Yaskawa INFORM job: DEMO_ROOF_UPPER_0625_3.JBI

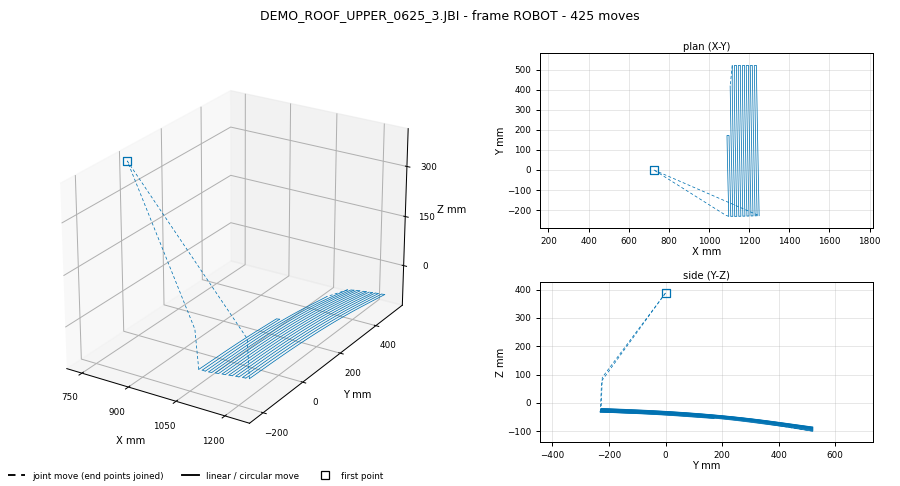
[picture p0: tool path of DEMO_ROOF_UPPER_0625_3.JBI in frame ROBOT, 425 of 425 moves have a stored position in this frame; points joined in program order, loops and branches not executed]
/JOB
//NAME DEMO_ROOF_UPPER_0625_3
//POS
///NPOS 425,0,0,0,0,0
///TOOL 0
///USER 0
///POSTYPE ROBOT
///RECTAN
///RCONF 1,0,0,0,0,0,0,0,0,0,0,0,0,0,0,0,0,0,0,0,0,0,0,0
C00000=725.000,0.000,388.500,-180.000,-0.000,0.000
///USER 0
///POSTYPE ROBOT
///RECTAN
C00001=1240.342,-223.716,89.889,177.727,-4.742,1.457
C00002=1249.517,-227.840,-19.446,177.737,-4.746,1.344
C00003=1247.381,-125.286,-23.774,177.737,-4.746,1.344
C00004=1246.860,-99.191,-24.873,177.524,-4.614,1.344
C00005=1246.366,-74.184,-26.020,177.315,-4.486,1.346
C00006=1245.874,-49.099,-27.262,177.100,-4.359,1.346
C00007=1245.386,-24.019,-28.598,176.878,-4.234,1.350
C00008=1244.921,0.054,-29.974,176.660,-4.119,1.352
C00009=1244.459,24.123,-31.441,176.435,-4.011,1.354
C00010=1244.000,48.187,-33.000,176.203,-3.911,1.356
C00011=1243.563,71.245,-34.588,175.975,-3.823,1.358
C00012=1243.128,94.298,-36.268,175.738,-3.746,1.364
C00013=1242.714,116.348,-37.962,175.506,-3.682,1.369
C00014=1242.302,138.394,-39.747,175.266,-3.631,1.372
C00015=1241.895,160.355,-41.616,175.018,-3.590,1.379
C00016=1241.506,181.391,-43.496,174.774,-3.563,1.388
C00017=1241.119,202.423,-45.465,174.522,-3.547,1.395
C00018=1240.735,223.453,-47.526,174.262,-3.543,1.405
C00019=1240.353,244.477,-49.679,173.998,-3.551,1.415
C00020=1239.993,264.406,-51.810,173.743,-3.570,1.430
C00021=1239.632,284.422,-54.040,173.482,-3.603,1.446
C00022=1239.273,304.436,-56.359,173.220,-3.652,1.464
C00023=1238.915,324.446,-58.768,172.960,-3.719,1.487
C00024=1238.558,344.452,-61.261,172.707,-3.804,1.516
C00025=1238.185,365.319,-63.950,172.464,-3.916,1.544
C00026=1237.775,388.282,-67.000,172.236,-4.061,1.575
C00027=1237.234,418.731,-71.176,172.012,-4.269,1.516
C00028=1235.598,520.410,-85.296,172.012,-4.269,1.516
C00029=1225.496,520.130,-86.161,172.024,-4.292,1.352
C00030=1227.173,414.926,-71.461,172.041,-4.257,1.444
C00031=1227.647,388.013,-67.749,172.243,-4.076,1.464
C00032=1228.055,365.054,-64.671,172.469,-3.926,1.465
C00033=1228.426,344.191,-61.961,172.711,-3.812,1.457
C00034=1228.783,324.187,-59.451,172.962,-3.723,1.446
C00035=1229.140,304.179,-57.031,173.222,-3.656,1.435
C00036=1229.498,284.168,-54.703,173.484,-3.606,1.425
C00037=1229.858,264.154,-52.466,173.744,-3.572,1.416
C00038=1230.218,244.226,-50.331,173.999,-3.552,1.409
C00039=1230.600,223.202,-48.173,174.262,-3.543,1.402
C00040=1230.984,202.174,-46.113,174.522,-3.547,1.397
C00041=1231.370,181.143,-44.146,174.773,-3.563,1.393
C00042=1231.759,160.106,-42.271,175.017,-3.589,1.390
C00043=1232.168,138.146,-40.407,175.265,-3.629,1.388
C00044=1232.580,116.100,-38.632,175.504,-3.681,1.387
C00045=1232.995,94.051,-36.947,175.737,-3.744,1.387
C00046=1233.430,70.997,-35.281,175.973,-3.821,1.388
C00047=1233.868,47.939,-33.708,176.201,-3.908,1.389
C00048=1234.328,23.876,-32.165,176.433,-4.009,1.390
C00049=1234.792,-0.193,-30.716,176.657,-4.117,1.392
C00050=1235.258,-24.267,-29.361,176.875,-4.232,1.394
C00051=1235.748,-49.347,-28.046,177.096,-4.356,1.396
C00052=1236.242,-74.432,-26.825,177.311,-4.484,1.398
C00053=1236.738,-99.438,-25.702,177.519,-4.611,1.401
C00054=1237.260,-125.533,-24.625,177.731,-4.744,1.408
C00055=1239.404,-228.090,-20.387,177.730,-4.743,1.421
C00056=1229.270,-228.359,-21.330,177.730,-4.743,1.425
C00057=1227.118,-125.798,-25.478,177.786,-4.870,1.350
C00058=1226.593,-99.702,-26.531,177.573,-4.744,1.353
C00059=1226.094,-74.695,-27.633,177.364,-4.620,1.354
C00060=1225.598,-49.609,-28.830,177.149,-4.498,1.356
C00061=1225.106,-24.527,-30.124,176.927,-4.377,1.357
C00062=1224.638,-0.451,-31.460,176.705,-4.267,1.363
C00063=1224.171,23.619,-32.889,176.477,-4.162,1.363
C00064=1223.729,46.685,-34.351,176.252,-4.070,1.369
C00065=1223.289,69.746,-35.904,176.019,-3.988,1.374
C00066=1222.851,92.801,-37.553,175.778,-3.915,1.379
C00067=1222.434,114.852,-39.224,175.541,-3.856,1.382
C00068=1222.021,136.900,-40.986,175.295,-3.808,1.391
C00069=1221.611,158.862,-42.838,175.043,-3.773,1.400
C00070=1221.220,179.899,-44.706,174.793,-3.751,1.405
C00071=1220.833,200.933,-46.665,174.536,-3.740,1.418
C00072=1220.447,221.963,-48.722,174.270,-3.742,1.425
C00073=1220.083,241.991,-50.773,174.013,-3.754,1.441
C00074=1219.721,261.920,-52.903,173.752,-3.778,1.453
C00075=1219.361,281.936,-55.137,173.484,-3.816,1.473
C00076=1219.002,301.949,-57.466,173.213,-3.868,1.492
C00077=1218.644,321.959,-59.890,172.942,-3.938,1.516
C00078=1218.290,341.844,-62.393,172.680,-4.027,1.546
C00079=1217.934,361.836,-64.998,172.432,-4.137,1.577
C00080=1217.544,383.804,-67.956,172.199,-4.283,1.605
C00081=1217.087,409.726,-71.548,172.001,-4.478,1.535
C00082=1215.344,520.125,-87.069,171.946,-4.534,1.543
C00083=1205.181,520.128,-88.023,171.968,-4.573,1.268
C00084=1206.771,418.484,-73.649,171.887,-4.817,1.451
C00085=1207.039,402.544,-71.393,171.980,-4.698,1.499
C00086=1207.480,377.609,-67.929,172.188,-4.502,1.531
C00087=1207.852,356.628,-65.100,172.432,-4.355,1.529
C00088=1208.208,336.632,-62.495,172.695,-4.241,1.517
C00089=1208.562,316.743,-59.999,172.970,-4.151,1.502
C00090=1208.902,297.725,-57.703,173.236,-4.082,1.487
C00091=1209.244,278.705,-55.496,173.500,-4.029,1.474
C00092=1209.605,258.687,-53.270,173.774,-3.986,1.462
C00093=1209.968,238.756,-51.147,174.040,-3.957,1.452
C00094=1210.333,218.726,-49.107,174.303,-3.939,1.443
C00095=1210.703,198.691,-47.158,174.560,-3.933,1.436
C00096=1211.092,177.657,-45.208,174.822,-3.938,1.429
C00097=1211.484,156.617,-43.353,175.077,-3.956,1.424
C00098=1211.876,135.651,-41.597,175.322,-3.985,1.420
C00099=1212.291,113.603,-39.846,175.572,-4.027,1.417
C00100=1212.710,91.550,-38.190,175.815,-4.081,1.415
C00101=1213.129,69.491,-36.627,176.049,-4.146,1.414
C00102=1213.572,46.429,-35.087,176.287,-4.225,1.413
C00103=1214.017,23.362,-33.642,176.515,-4.312,1.413
C00104=1214.485,-0.710,-32.229,176.746,-4.411,1.413
C00105=1214.956,-24.788,-30.913,176.969,-4.517,1.413
C00106=1215.450,-49.871,-29.640,177.193,-4.632,1.413
C00107=1215.949,-74.960,-28.463,177.409,-4.751,1.413
C00108=1216.450,-99.968,-27.384,177.617,-4.870,1.414
C00109=1216.979,-126.065,-26.352,177.828,-4.992,1.419
C00110=1219.138,-228.629,-22.291,177.826,-4.991,1.444
C00111=1209.008,-228.900,-23.270,177.826,-4.991,1.443
C00112=1206.841,-126.333,-27.248,177.879,-5.116,1.364
C00113=1206.310,-100.234,-28.259,177.669,-5.000,1.368
C00114=1205.806,-75.226,-29.318,177.461,-4.886,1.369
C00115=1205.305,-50.136,-30.474,177.243,-4.772,1.374
C00116=1204.828,-26.050,-31.675,177.025,-4.666,1.379
C00117=1204.354,-1.971,-32.970,176.800,-4.564,1.383
C00118=1203.883,22.103,-34.360,176.566,-4.469,1.387
C00119=1203.437,45.172,-35.787,176.333,-4.386,1.393
C00120=1202.992,68.236,-37.309,176.092,-4.312,1.401
C00121=1202.570,90.296,-38.858,175.853,-4.252,1.406
C00122=1202.151,112.351,-40.500,175.605,-4.202,1.416
C00123=1201.754,133.325,-42.153,175.362,-4.166,1.425
C00124=1201.358,154.370,-43.902,175.109,-4.140,1.431
C00125=1200.965,175.412,-45.745,174.849,-4.127,1.446
C00126=1200.593,195.451,-47.592,174.595,-4.125,1.458
C00127=1200.223,215.487,-49.529,174.332,-4.134,1.469
C00128=1199.857,235.428,-51.549,174.065,-4.155,1.487
C00129=1199.492,255.451,-53.673,173.791,-4.189,1.502
C00130=1199.148,274.476,-55.782,173.525,-4.233,1.522
C00131=1198.805,293.499,-57.981,173.254,-4.290,1.542
C00132=1198.467,312.407,-60.256,172.981,-4.359,1.566
C00133=1198.129,331.416,-62.637,172.707,-4.443,1.595
C00134=1197.791,350.423,-65.107,172.439,-4.546,1.631
C00135=1197.436,370.419,-67.800,172.178,-4.681,1.666
C00136=1197.033,393.235,-70.973,171.954,-4.868,1.663
C00137=1196.606,418.506,-74.570,171.896,-5.210,0.598
C00138=1196.859,520.156,-88.981,171.896,-5.210,0.598
C00139=1185.350,520.147,-90.183,171.840,-5.121,1.226
C00140=1186.488,414.926,-75.019,171.764,-5.333,1.478
C00141=1186.975,387.040,-71.024,171.921,-5.087,1.597
C00142=1187.346,366.069,-68.096,172.154,-4.905,1.611
C00143=1187.680,347.197,-65.546,172.420,-4.773,1.598
C00144=1188.016,328.188,-63.070,172.699,-4.668,1.577
C00145=1188.354,309.176,-60.689,172.981,-4.580,1.556
C00146=1188.693,290.267,-58.414,173.261,-4.507,1.537
C00147=1189.036,271.241,-56.218,173.539,-4.445,1.521
C00148=1189.382,252.214,-54.115,173.810,-4.395,1.506
C00149=1189.730,233.186,-52.101,174.075,-4.358,1.494
C00150=1190.096,213.243,-50.085,174.348,-4.332,1.483
C00151=1190.467,193.206,-48.155,174.615,-4.317,1.473
C00152=1190.841,173.165,-46.317,174.876,-4.314,1.465
C00153=1191.236,152.122,-44.485,175.140,-4.323,1.458
C00154=1191.632,131.074,-42.747,175.397,-4.344,1.452
C00155=1192.031,110.099,-41.110,175.644,-4.376,1.448
C00156=1192.452,88.042,-39.484,175.896,-4.421,1.444
C00157=1192.876,65.980,-37.954,176.139,-4.478,1.441
C00158=1193.303,43.913,-36.516,176.374,-4.544,1.439
C00159=1193.753,20.842,-35.107,176.609,-4.622,1.437
C00160=1194.206,-2.233,-33.792,176.837,-4.709,1.436
C00161=1194.682,-26.315,-32.515,177.064,-4.805,1.434
C00162=1195.161,-50.401,-31.332,177.283,-4.907,1.432
C00163=1195.666,-75.492,-30.196,177.501,-5.015,1.429
C00164=1196.172,-100.503,-29.156,177.708,-5.124,1.427
C00165=1196.706,-126.601,-28.166,177.916,-5.236,1.429
C00166=1198.879,-229.172,-24.267,177.913,-5.235,1.461
C00167=1188.753,-229.444,-25.281,177.913,-5.235,1.460
C00168=1186.572,-126.871,-29.104,177.963,-5.358,1.376
C00169=1186.036,-100.771,-30.076,177.755,-5.252,1.382
C00170=1185.505,-74.676,-31.143,177.538,-5.144,1.388
C00171=1185.000,-49.668,-32.262,177.320,-5.042,1.390
C00172=1184.518,-25.580,-33.431,177.099,-4.945,1.398
C00173=1184.040,-1.497,-34.695,176.867,-4.854,1.405
C00174=1183.585,21.581,-36.000,176.637,-4.773,1.412
C00175=1183.133,44.653,-37.399,176.396,-4.700,1.418
C00176=1182.705,66.720,-38.830,176.157,-4.638,1.426
C00177=1182.279,88.784,-40.356,175.907,-4.587,1.436
C00178=1181.875,109.842,-41.903,175.662,-4.548,1.446
C00179=1181.476,130.820,-43.536,175.408,-4.521,1.457
C00180=1181.078,151.868,-45.269,175.145,-4.504,1.470
C00181=1180.701,171.914,-47.012,174.886,-4.501,1.482
C00182=1180.327,191.956,-48.847,174.620,-4.508,1.499
C00183=1179.954,211.995,-50.776,174.347,-4.527,1.514
C00184=1179.587,231.939,-52.792,174.068,-4.558,1.534
C00185=1179.238,250.968,-54.809,173.794,-4.601,1.553
C00186=1178.892,269.996,-56.918,173.516,-4.656,1.575
C00187=1178.550,288.915,-59.108,173.233,-4.724,1.597
C00188=1178.210,307.932,-61.405,172.945,-4.802,1.626
C00189=1177.871,326.944,-63.798,172.654,-4.893,1.654
C00190=1177.553,344.962,-66.156,172.378,-4.993,1.685
C00191=1177.239,362.842,-68.583,172.105,-5.112,1.733
C00192=1176.903,381.834,-71.249,171.861,-5.277,1.755
C00193=1176.285,417.612,-76.422,171.776,-5.762,0.547
C00194=1176.794,520.192,-91.175,171.773,-5.768,0.548
C00195=1167.129,520.224,-92.309,171.773,-5.768,0.548
C00196=1166.131,417.999,-77.542,171.608,-5.896,1.543
C00197=1166.415,400.557,-74.981,171.644,-5.743,1.638
C00198=1166.870,374.642,-71.222,171.849,-5.468,1.719
C00199=1167.168,357.627,-68.832,172.107,-5.327,1.712
C00200=1167.484,339.616,-66.391,172.394,-5.210,1.674
C00201=1167.800,321.721,-64.055,172.677,-5.108,1.638
C00202=1168.121,303.700,-61.792,172.959,-5.019,1.610
C00203=1168.444,285.678,-59.617,173.238,-4.939,1.587
C00204=1168.787,266.757,-57.429,173.525,-4.866,1.568
C00205=1169.134,247.727,-55.324,173.810,-4.805,1.550
C00206=1169.483,228.695,-53.313,174.089,-4.758,1.535
C00207=1169.835,209.660,-51.394,174.360,-4.723,1.522
C00208=1170.206,189.708,-49.479,174.637,-4.698,1.510
C00209=1170.581,169.664,-47.651,174.909,-4.686,1.500
C00210=1170.960,149.616,-45.918,175.172,-4.686,1.492
C00211=1171.341,129.564,-44.275,175.427,-4.697,1.485
C00212=1171.741,108.585,-42.651,175.686,-4.720,1.479
C00213=1172.147,87.526,-41.114,175.936,-4.754,1.474
C00214=1172.574,65.461,-39.602,176.189,-4.801,1.469
C00215=1173.005,43.391,-38.185,176.432,-4.857,1.466
C00216=1173.438,21.317,-36.860,176.665,-4.923,1.463
C00217=1173.896,-1.762,-35.569,176.899,-4.999,1.460
C00218=1174.376,-25.846,-34.321,177.132,-5.085,1.456
C00219=1174.860,-49.935,-33.167,177.354,-5.176,1.452
C00220=1175.368,-74.945,-32.067,177.574,-5.273,1.445
C00221=1175.902,-101.040,-31.018,177.791,-5.375,1.437
C00222=1176.441,-127.141,-30.065,177.997,-5.475,1.435
C00223=1178.628,-229.716,-26.314,177.992,-5.474,1.477
C00224=1168.506,-229.991,-27.362,177.993,-5.474,1.476
C00225=1166.312,-127.413,-31.046,178.037,-5.595,1.392
C00226=1165.770,-101.311,-31.982,177.834,-5.502,1.397
C00227=1165.233,-75.213,-33.014,177.617,-5.406,1.403
C00228=1164.723,-50.204,-34.098,177.396,-5.315,1.409
C00229=1164.236,-26.114,-35.235,177.172,-5.229,1.417
C00230=1163.773,-3.028,-36.417,176.946,-5.152,1.423
C00231=1163.315,20.053,-37.690,176.708,-5.081,1.435
C00232=1162.878,42.128,-39.000,176.472,-5.019,1.441
C00233=1162.446,64.199,-40.404,176.225,-4.967,1.452
C00234=1162.036,85.266,-41.833,175.978,-4.926,1.464
C00235=1161.631,106.252,-43.350,175.723,-4.895,1.476
C00236=1161.227,127.308,-44.967,175.459,-4.875,1.489
C00237=1160.845,147.362,-46.600,175.198,-4.867,1.504
C00238=1160.465,167.411,-48.325,174.930,-4.871,1.519
C00239=1160.089,187.456,-50.145,174.651,-4.887,1.538
C00240=1159.735,206.413,-51.959,174.382,-4.914,1.555
C00241=1159.383,225.450,-53.870,174.104,-4.952,1.578
C00242=1159.032,244.484,-55.875,173.819,-5.004,1.598
C00243=1158.685,263.516,-57.978,173.528,-5.068,1.622
C00244=1158.514,272.977,-59.059,173.380,-5.104,1.639
C00245=1158.180,291.450,-61.241,173.091,-5.184,1.665
C00246=1157.858,309.475,-63.461,172.805,-5.273,1.694
C00247=1157.539,327.433,-65.765,172.515,-5.374,1.728
C00248=1157.223,345.387,-68.159,172.223,-5.489,1.758
C00249=1156.918,362.904,-70.585,171.931,-5.612,1.800
C00250=1156.770,371.414,-71.796,171.788,-5.679,1.832
C00251=1156.441,390.250,-74.544,171.563,-5.872,1.858
C00252=1155.996,416.130,-78.380,171.597,-6.236,1.004
C00253=1155.842,520.246,-93.672,171.591,-6.255,1.007
C00254=1145.788,520.287,-94.973,171.591,-6.255,1.007
C00255=1145.854,415.867,-79.499,171.450,-6.413,1.614
C00256=1146.399,384.053,-74.735,171.500,-6.064,1.847
C00257=1146.689,367.188,-72.266,171.746,-5.876,2.037
C00258=1146.984,350.164,-69.859,172.056,-5.767,1.850
C00259=1147.299,332.149,-67.408,172.367,-5.650,1.740
C00260=1147.617,314.134,-65.052,172.667,-5.539,1.689
C00261=1147.937,296.227,-62.803,172.960,-5.439,1.656
C00262=1148.261,278.200,-60.632,173.251,-5.351,1.630
C00263=1148.588,260.172,-58.552,173.536,-5.275,1.609
C00264=1148.916,242.235,-56.572,173.817,-5.210,1.591
C00265=1149.267,223.200,-54.565,174.107,-5.153,1.574
C00266=1149.620,204.162,-52.655,174.391,-5.108,1.559
C00267=1149.975,185.203,-50.846,174.666,-5.077,1.546
C00268=1150.333,166.155,-49.120,174.934,-5.057,1.535
C00269=1150.714,146.104,-47.397,175.209,-5.048,1.525
C00270=1151.097,126.049,-45.770,175.475,-5.051,1.517
C00271=1151.483,105.990,-44.235,175.731,-5.065,1.510
C00272=1151.889,85.004,-42.723,175.991,-5.091,1.504
C00273=1152.300,63.935,-41.299,176.241,-5.127,1.499
C00274=1152.734,41.863,-39.905,176.492,-5.175,1.495
C00275=1153.172,19.786,-38.604,176.732,-5.231,1.491
C00276=1153.633,-3.296,-37.343,176.972,-5.297,1.487
C00277=1154.099,-26.382,-36.175,177.200,-5.369,1.482
C00278=1154.588,-50.474,-35.052,177.425,-5.449,1.475
C00279=1155.101,-75.485,-33.984,177.646,-5.535,1.463
C00280=1155.640,-101.584,-32.968,177.865,-5.625,1.440
C00281=1158.386,-230.265,-28.426,178.062,-5.709,1.493
C00282=1148.266,-230.540,-29.499,178.062,-5.709,1.493
C00283=1145.491,-100.855,-34.013,177.892,-5.746,1.412
C00284=1144.949,-74.756,-35.017,177.676,-5.664,1.420
C00285=1144.432,-49.661,-36.079,177.452,-5.585,1.427
C00286=1143.943,-25.652,-37.189,177.226,-5.511,1.438
C00287=1143.475,-2.564,-38.349,176.995,-5.445,1.446
C00288=1143.012,20.519,-39.604,176.752,-5.384,1.455
C00289=1142.574,42.597,-40.898,176.506,-5.333,1.468
C00290=1142.158,63.671,-42.224,176.261,-5.293,1.479
C00291=1141.745,84.740,-43.642,176.005,-5.261,1.491
C00292=1141.337,105.728,-45.150,175.740,-5.239,1.509
C00293=1140.950,125.788,-46.684,175.477,-5.228,1.522
C00294=1140.566,145.843,-48.311,175.204,-5.229,1.540
C00295=1140.203,164.897,-49.947,174.937,-5.242,1.554
C00296=1139.846,183.863,-51.666,174.662,-5.265,1.579
C00297=1139.489,202.905,-53.484,174.379,-5.301,1.600
C00298=1139.135,221.945,-55.399,174.089,-5.350,1.621
C00299=1138.803,239.984,-57.303,173.806,-5.408,1.649
C00300=1138.474,257.922,-59.286,173.520,-5.476,1.673
C00301=1138.148,275.951,-61.370,173.226,-5.556,1.703
C00302=1137.824,293.980,-63.549,172.929,-5.647,1.736
C00303=1137.504,311.887,-65.806,172.628,-5.751,1.769
C00304=1137.186,329.904,-68.174,172.321,-5.870,1.807
C00305=1136.889,346.927,-70.501,172.026,-5.997,1.848
C00306=1136.561,365.850,-73.192,170.935,-4.967,9.690
C00307=1136.241,367.898,-73.529,171.563,-7.814,2.067
C00308=1135.959,385.991,-76.231,171.299,-7.828,2.160
C00309=1135.521,412.147,-80.220,171.226,-8.092,2.030
C00310=1135.442,417.940,-81.106,171.435,-8.424,0.545
C00311=1136.727,520.330,-96.358,171.435,-8.442,0.548
C00312=1126.382,520.298,-98.281,171.435,-8.442,0.548
C00313=1125.381,417.119,-82.483,171.049,-8.208,1.827
C00314=1125.602,403.547,-80.368,171.147,-7.985,1.913
C00315=1125.823,389.970,-78.279,171.250,-7.865,2.012
C00316=1126.065,374.394,-75.927,171.430,-7.802,2.184
C00317=1126.339,356.814,-73.353,171.721,-7.788,2.189
C00318=1126.620,339.218,-70.870,172.041,-7.789,2.024
C00319=1126.921,320.897,-68.382,172.348,-7.768,1.959
C00320=1127.232,302.284,-65.952,172.653,-7.738,1.921
C00321=1127.550,283.660,-63.620,172.954,-7.704,1.893
C00322=1127.870,265.300,-61.419,173.249,-7.660,1.868
C00323=1128.204,246.649,-59.279,173.566,-7.606,1.843
C00324=1128.543,227.991,-57.233,173.857,-7.542,1.819
C00325=1128.905,208.607,-55.213,174.137,-7.447,1.792
C00326=1129.220,191.922,-53.554,174.405,-7.376,1.771
C00327=1129.581,173.239,-51.782,174.683,-7.283,1.747
C00328=1129.943,154.819,-50.124,174.969,-7.174,1.724
C00329=1130.322,136.119,-48.537,175.244,-7.030,1.700
C00330=1130.746,115.453,-46.876,175.516,-6.871,1.673
C00331=1131.117,109.456,-46.393,175.690,-5.408,1.547
C00332=1131.233,103.465,-45.949,175.769,-5.410,1.545
C00333=1131.622,83.476,-44.522,176.025,-5.427,1.538
C00334=1132.037,62.405,-43.113,176.284,-5.454,1.533
C00335=1132.454,41.330,-41.798,176.532,-5.490,1.530
C00336=1132.895,19.251,-40.517,176.779,-5.536,1.526
C00337=1133.340,-2.834,-39.328,177.014,-5.589,1.522
C00338=1133.810,-25.924,-38.179,177.247,-5.650,1.517
C00339=1134.302,-49.932,-37.081,177.475,-5.717,1.509
C00340=1134.822,-75.029,-36.032,177.700,-5.791,1.492
C00341=1135.366,-101.128,-35.042,177.921,-5.869,1.434
C00342=1138.150,-230.816,-30.596,178.120,-5.942,1.511
C00343=1128.042,-231.097,-31.847,178.120,-5.942,1.511
C00344=1125.676,-121.895,-35.392,178.488,-6.151,-2.162
C00345=1125.946,-115.292,-35.577,178.155,-3.671,1.544
C00346=1125.370,-92.063,-36.372,177.929,-4.083,1.563
C00347=1124.818,-69.593,-37.223,177.704,-4.483,1.569
C00348=1124.294,-47.851,-38.141,177.466,-4.842,1.578
C00349=1123.858,-29.386,-38.992,177.244,-5.124,1.594
C00350=1123.374,-8.652,-40.025,177.013,-5.431,1.614
C00351=1122.879,12.802,-41.185,176.768,-5.737,1.631
C00352=1122.433,32.530,-42.335,176.521,-5.997,1.644
C00353=1121.981,52.975,-43.617,176.261,-6.237,1.663
C00354=1121.532,73.692,-45.012,175.992,-6.461,1.690
C00355=1121.074,95.121,-46.552,175.724,-6.683,1.711
C00356=1120.683,113.831,-47.986,175.448,-6.849,1.728
C00357=1120.267,134.248,-49.649,175.176,-7.005,1.762
C00358=1119.870,153.937,-51.342,174.902,-7.159,1.778
C00359=1119.523,171.627,-52.949,174.639,-7.266,1.795
C00360=1119.170,190.024,-54.704,174.372,-7.360,1.820
C00361=1118.837,207.698,-56.471,174.100,-7.436,1.851
C00362=1118.487,226.442,-58.435,173.823,-7.527,1.871
C00363=1118.156,244.731,-60.446,173.537,-7.590,1.898
C00364=1117.823,263.373,-62.587,173.246,-7.648,1.918
C00365=1117.517,281.010,-64.699,172.965,-7.692,1.944
C00366=1117.204,299.349,-66.989,172.669,-7.725,1.970
C00367=1116.892,317.958,-69.410,172.367,-7.757,1.993
C00368=1116.604,335.560,-71.792,172.081,-7.783,2.017
C00369=1116.311,353.861,-74.362,171.777,-7.806,2.037
C00370=1116.038,371.439,-76.925,171.478,-7.816,2.067
C00371=1115.783,388.010,-79.424,171.208,-7.834,2.148
C00372=1115.471,407.391,-82.438,170.932,-7.975,2.250
C00373=1115.339,415.169,-83.674,170.972,-8.268,1.170
C00374=1115.600,520.260,-100.242,170.917,-8.338,1.182
C00375=1105.173,418.619,-83.928,170.917,-8.338,1.182
C00376=1107.147,298.116,-68.243,172.672,-7.731,1.901
C00377=1107.459,279.788,-65.952,172.965,-7.695,1.877
C00378=1107.783,261.161,-63.719,173.255,-7.647,1.854
C00379=1108.097,243.522,-61.690,173.521,-7.591,1.833
C00380=1108.430,225.162,-59.665,173.796,-7.524,1.810
C00381=1108.757,207.503,-57.799,174.068,-7.439,1.787
C00382=1109.107,188.839,-55.921,174.343,-7.357,1.763
C00383=1109.478,169.456,-54.061,174.616,-7.256,1.737
C00384=1109.844,150.777,-52.354,174.879,-7.137,1.719
C00385=1110.254,130.379,-50.586,175.152,-6.977,1.694
C00386=1110.675,109.690,-48.891,175.427,-6.815,1.669
C00387=1111.080,90.273,-47.391,175.688,-6.633,1.644
C00388=1111.542,68.573,-45.811,175.954,-6.405,1.616
C00389=1111.984,48.145,-44.418,176.210,-6.179,1.595
C00390=1112.440,27.431,-43.097,176.458,-5.929,1.570
C00391=1112.901,6.994,-41.877,176.695,-5.648,1.544
C00392=1113.399,-14.729,-40.672,176.944,-5.339,1.515
C00393=1113.920,-37.176,-39.523,177.184,-5.006,1.484
C00394=1114.474,-60.628,-38.422,177.428,-4.627,1.447
C00395=1114.974,-81.365,-37.532,177.663,-4.268,1.403
C00396=1115.570,-105.823,-36.579,177.890,-3.838,1.299
C00397=1116.126,-128.289,-35.789,178.122,-3.423,1.156
C00398=1118.329,-230.871,-32.208,178.112,-3.418,1.325
C00399=1108.146,-230.595,-32.508,178.112,-3.418,1.326
C00400=1105.973,-128.024,-36.412,177.896,-3.401,1.531
C00401=1105.498,-108.575,-37.156,177.715,-3.765,1.538
C00402=1104.909,-84.129,-38.176,177.492,-4.199,1.559
C00403=1104.390,-62.401,-39.167,177.269,-4.581,1.571
C00404=1103.840,-38.963,-40.329,177.040,-4.963,1.584
C00405=1103.324,-16.528,-41.530,176.804,-5.297,1.605
C00406=1102.832,5.188,-42.783,176.558,-5.608,1.631
C00407=1102.352,26.611,-44.110,176.325,-5.905,1.646
C00408=1101.877,48.315,-45.542,176.080,-6.170,1.664
C00409=1101.434,68.944,-46.992,175.842,-6.405,1.569
C00410=1099.434,171.341,-54.166,175.842,-6.405,1.569
C00411=1089.364,171.048,-55.496,175.842,-6.405,1.569
C00412=1091.343,68.664,-48.124,175.837,-6.402,1.616
C00413=1091.781,48.041,-46.635,176.088,-6.174,1.595
C00414=1092.250,26.345,-45.156,176.333,-5.910,1.570
C00415=1092.724,4.927,-43.776,176.567,-5.613,1.542
C00416=1093.212,-16.785,-42.468,176.813,-5.302,1.513
C00417=1093.722,-39.214,-41.207,177.049,-4.968,1.481
C00418=1094.266,-62.649,-39.979,177.279,-4.587,1.443
C00419=1094.779,-84.373,-38.919,177.504,-4.206,1.400
C00420=1095.364,-108.816,-37.822,177.728,-3.773,1.339
C00421=1095.835,-128.264,-37.017,177.910,-3.409,1.296
C00422=1097.987,-230.821,-32.791,177.908,-3.408,1.326
C00423=1084.082,-226.185,76.923,177.907,-3.408,1.347
///USER 0
///POSTYPE ROBOT
///RECTAN
C00424=725.000,0.000,388.500,-180.000,-0.000,0.000
//INST
///DATE 2021/06/25 11:33
///ATTR SC,RW,RJ
////FRAME ROBOT
///GROUP1 RB1
NOP
MOVJ C00000 VJ=25.00 PL=0
'Path Start: roof
MOVJ C00001 VJ=25.00 PL=0
MOVJ C00002 VJ=25.00 PL=0
SPYON
MOVL C00003 V=800.0 PL=8
MOVL C00004 V=800.0 PL=8
MOVL C00005 V=800.0 PL=8
MOVL C00006 V=800.0 PL=8
MOVL C00007 V=800.0 PL=8
MOVL C00008 V=800.0 PL=8
MOVL C00009 V=800.0 PL=8
MOVL C00010 V=800.0 PL=8
MOVL C00011 V=800.0 PL=8
MOVL C00012 V=800.0 PL=8
MOVL C00013 V=800.0 PL=8
MOVL C00014 V=800.0 PL=8
MOVL C00015 V=800.0 PL=8
MOVL C00016 V=800.0 PL=8
MOVL C00017 V=800.0 PL=8
MOVL C00018 V=800.0 PL=8
MOVL C00019 V=800.0 PL=8
MOVL C00020 V=800.0 PL=8
MOVL C00021 V=800.0 PL=8
MOVL C00022 V=800.0 PL=8
MOVL C00023 V=800.0 PL=8
MOVL C00024 V=800.0 PL=8
MOVL C00025 V=800.0 PL=8
MOVL C00026 V=800.0 PL=8
MOVL C00027 V=800.0 PL=8
MOVL C00028 V=800.0 PL=0
SPYOF
MOVJ C00029 VJ=25.00 PL=0
SPYON
MOVL C00030 V=800.0 PL=8
MOVL C00031 V=800.0 PL=8
MOVL C00032 V=800.0 PL=8
MOVL C00033 V=800.0 PL=8
MOVL C00034 V=800.0 PL=8
MOVL C00035 V=800.0 PL=8
MOVL C00036 V=800.0 PL=8
MOVL C00037 V=800.0 PL=8
MOVL C00038 V=800.0 PL=8
MOVL C00039 V=800.0 PL=8
MOVL C00040 V=800.0 PL=8
MOVL C00041 V=800.0 PL=8
MOVL C00042 V=800.0 PL=8
MOVL C00043 V=800.0 PL=8
MOVL C00044 V=800.0 PL=8
MOVL C00045 V=800.0 PL=8
MOVL C00046 V=800.0 PL=8
MOVL C00047 V=800.0 PL=8
MOVL C00048 V=800.0 PL=8
MOVL C00049 V=800.0 PL=8
MOVL C00050 V=800.0 PL=8
MOVL C00051 V=800.0 PL=8
MOVL C00052 V=800.0 PL=8
MOVL C00053 V=800.0 PL=8
MOVL C00054 V=800.0 PL=8
MOVL C00055 V=800.0 PL=0
SPYOF
MOVJ C00056 VJ=25.00 PL=0
SPYON
MOVL C00057 V=800.0 PL=8
MOVL C00058 V=800.0 PL=8
MOVL C00059 V=800.0 PL=8
MOVL C00060 V=800.0 PL=8
MOVL C00061 V=800.0 PL=8
MOVL C00062 V=800.0 PL=8
MOVL C00063 V=800.0 PL=8
MOVL C00064 V=800.0 PL=8
MOVL C00065 V=800.0 PL=8
MOVL C00066 V=800.0 PL=8
MOVL C00067 V=800.0 PL=8
MOVL C00068 V=800.0 PL=8
MOVL C00069 V=800.0 PL=8
MOVL C00070 V=800.0 PL=8
MOVL C00071 V=800.0 PL=8
MOVL C00072 V=800.0 PL=8
MOVL C00073 V=800.0 PL=8
MOVL C00074 V=800.0 PL=8
MOVL C00075 V=800.0 PL=8
MOVL C00076 V=800.0 PL=8
MOVL C00077 V=800.0 PL=8
MOVL C00078 V=800.0 PL=8
MOVL C00079 V=800.0 PL=8
MOVL C00080 V=800.0 PL=8
MOVL C00081 V=800.0 PL=8
MOVL C00082 V=800.0 PL=0
SPYOF
MOVJ C00083 VJ=25.00 PL=0
SPYON
MOVL C00084 V=800.0 PL=8
MOVL C00085 V=800.0 PL=8
MOVL C00086 V=800.0 PL=8
MOVL C00087 V=800.0 PL=8
MOVL C00088 V=800.0 PL=8
MOVL C00089 V=800.0 PL=8
MOVL C00090 V=800.0 PL=8
MOVL C00091 V=800.0 PL=8
MOVL C00092 V=800.0 PL=8
MOVL C00093 V=800.0 PL=8
MOVL C00094 V=800.0 PL=8
MOVL C00095 V=800.0 PL=8
MOVL C00096 V=800.0 PL=8
MOVL C00097 V=800.0 PL=8
MOVL C00098 V=800.0 PL=8
MOVL C00099 V=800.0 PL=8
MOVL C00100 V=800.0 PL=8
MOVL C00101 V=800.0 PL=8
MOVL C00102 V=800.0 PL=8
MOVL C00103 V=800.0 PL=8
MOVL C00104 V=800.0 PL=8
MOVL C00105 V=800.0 PL=8
MOVL C00106 V=800.0 PL=8
MOVL C00107 V=800.0 PL=8
MOVL C00108 V=800.0 PL=8
MOVL C00109 V=800.0 PL=8
MOVL C00110 V=800.0 PL=0
SPYOF
MOVJ C00111 VJ=25.00 PL=0
SPYON
MOVL C00112 V=800.0 PL=8
MOVL C00113 V=800.0 PL=8
MOVL C00114 V=800.0 PL=8
MOVL C00115 V=800.0 PL=8
MOVL C00116 V=800.0 PL=8
MOVL C00117 V=800.0 PL=8
MOVL C00118 V=800.0 PL=8
MOVL C00119 V=800.0 PL=8
MOVL C00120 V=800.0 PL=8
MOVL C00121 V=800.0 PL=8
MOVL C00122 V=800.0 PL=8
MOVL C00123 V=800.0 PL=8
MOVL C00124 V=800.0 PL=8
MOVL C00125 V=800.0 PL=8
MOVL C00126 V=800.0 PL=8
MOVL C00127 V=800.0 PL=8
MOVL C00128 V=800.0 PL=8
MOVL C00129 V=800.0 PL=8
MOVL C00130 V=800.0 PL=8
MOVL C00131 V=800.0 PL=8
MOVL C00132 V=800.0 PL=8
MOVL C00133 V=800.0 PL=8
MOVL C00134 V=800.0 PL=8
MOVL C00135 V=800.0 PL=8
MOVL C00136 V=800.0 PL=8
MOVL C00137 V=800.0 PL=8
MOVL C00138 V=800.0 PL=0
SPYOF
MOVJ C00139 VJ=25.00 PL=0
SPYON
MOVL C00140 V=800.0 PL=8
MOVL C00141 V=800.0 PL=8
MOVL C00142 V=800.0 PL=8
MOVL C00143 V=800.0 PL=8
MOVL C00144 V=800.0 PL=8
MOVL C00145 V=800.0 PL=8
MOVL C00146 V=800.0 PL=8
MOVL C00147 V=800.0 PL=8
MOVL C00148 V=800.0 PL=8
MOVL C00149 V=800.0 PL=8
MOVL C00150 V=800.0 PL=8
MOVL C00151 V=800.0 PL=8
MOVL C00152 V=800.0 PL=8
MOVL C00153 V=800.0 PL=8
MOVL C00154 V=800.0 PL=8
MOVL C00155 V=800.0 PL=8
MOVL C00156 V=800.0 PL=8
MOVL C00157 V=800.0 PL=8
MOVL C00158 V=800.0 PL=8
MOVL C00159 V=800.0 PL=8
MOVL C00160 V=800.0 PL=8
MOVL C00161 V=800.0 PL=8
MOVL C00162 V=800.0 PL=8
MOVL C00163 V=800.0 PL=8
MOVL C00164 V=800.0 PL=8
MOVL C00165 V=800.0 PL=8
MOVL C00166 V=800.0 PL=0
SPYOF
MOVJ C00167 VJ=25.00 PL=0
SPYON
MOVL C00168 V=800.0 PL=8
MOVL C00169 V=800.0 PL=8
MOVL C00170 V=800.0 PL=8
MOVL C00171 V=800.0 PL=8
MOVL C00172 V=800.0 PL=8
MOVL C00173 V=800.0 PL=8
MOVL C00174 V=800.0 PL=8
MOVL C00175 V=800.0 PL=8
MOVL C00176 V=800.0 PL=8
MOVL C00177 V=800.0 PL=8
MOVL C00178 V=800.0 PL=8
MOVL C00179 V=800.0 PL=8
MOVL C00180 V=800.0 PL=8
MOVL C00181 V=800.0 PL=8
MOVL C00182 V=800.0 PL=8
MOVL C00183 V=800.0 PL=8
MOVL C00184 V=800.0 PL=8
MOVL C00185 V=800.0 PL=8
MOVL C00186 V=800.0 PL=8
MOVL C00187 V=800.0 PL=8
MOVL C00188 V=800.0 PL=8
MOVL C00189 V=800.0 PL=8
MOVL C00190 V=800.0 PL=8
MOVL C00191 V=800.0 PL=8
MOVL C00192 V=800.0 PL=8
MOVL C00193 V=800.0 PL=8
MOVL C00194 V=800.0 PL=0
SPYOF
MOVJ C00195 VJ=25.00 PL=0
SPYON
MOVL C00196 V=800.0 PL=8
MOVL C00197 V=800.0 PL=8
MOVL C00198 V=800.0 PL=8
MOVL C00199 V=800.0 PL=8
MOVL C00200 V=800.0 PL=8
MOVL C00201 V=800.0 PL=8
MOVL C00202 V=800.0 PL=8
MOVL C00203 V=800.0 PL=8
MOVL C00204 V=800.0 PL=8
MOVL C00205 V=800.0 PL=8
MOVL C00206 V=800.0 PL=8
MOVL C00207 V=800.0 PL=8
MOVL C00208 V=800.0 PL=8
MOVL C00209 V=800.0 PL=8
MOVL C00210 V=800.0 PL=8
MOVL C00211 V=800.0 PL=8
MOVL C00212 V=800.0 PL=8
MOVL C00213 V=800.0 PL=8
MOVL C00214 V=800.0 PL=8
MOVL C00215 V=800.0 PL=8
MOVL C00216 V=800.0 PL=8
MOVL C00217 V=800.0 PL=8
MOVL C00218 V=800.0 PL=8
MOVL C00219 V=800.0 PL=8
MOVL C00220 V=800.0 PL=8
MOVL C00221 V=800.0 PL=8
MOVL C00222 V=800.0 PL=8
MOVL C00223 V=800.0 PL=0
SPYOF
MOVJ C00224 VJ=25.00 PL=0
SPYON
MOVL C00225 V=800.0 PL=8
MOVL C00226 V=800.0 PL=8
MOVL C00227 V=800.0 PL=8
MOVL C00228 V=800.0 PL=8
MOVL C00229 V=800.0 PL=8
MOVL C00230 V=800.0 PL=8
MOVL C00231 V=800.0 PL=8
MOVL C00232 V=800.0 PL=8
MOVL C00233 V=800.0 PL=8
MOVL C00234 V=800.0 PL=8
MOVL C00235 V=800.0 PL=8
MOVL C00236 V=800.0 PL=8
MOVL C00237 V=800.0 PL=8
MOVL C00238 V=800.0 PL=8
MOVL C00239 V=800.0 PL=8
MOVL C00240 V=800.0 PL=8
MOVL C00241 V=800.0 PL=8
MOVL C00242 V=800.0 PL=8
MOVL C00243 V=800.0 PL=8
MOVL C00244 V=800.0 PL=8
MOVL C00245 V=800.0 PL=8
MOVL C00246 V=800.0 PL=8
MOVL C00247 V=800.0 PL=8
MOVL C00248 V=800.0 PL=8
MOVL C00249 V=800.0 PL=8
MOVL C00250 V=800.0 PL=8
MOVL C00251 V=800.0 PL=8
MOVL C00252 V=800.0 PL=8
MOVL C00253 V=800.0 PL=0
SPYOF
MOVJ C00254 VJ=25.00 PL=0
SPYON
MOVL C00255 V=800.0 PL=8
MOVL C00256 V=800.0 PL=8
MOVL C00257 V=800.0 PL=8
MOVL C00258 V=800.0 PL=8
MOVL C00259 V=800.0 PL=8
MOVL C00260 V=800.0 PL=8
MOVL C00261 V=800.0 PL=8
MOVL C00262 V=800.0 PL=8
MOVL C00263 V=800.0 PL=8
MOVL C00264 V=800.0 PL=8
MOVL C00265 V=800.0 PL=8
MOVL C00266 V=800.0 PL=8
MOVL C00267 V=800.0 PL=8
MOVL C00268 V=800.0 PL=8
MOVL C00269 V=800.0 PL=8
MOVL C00270 V=800.0 PL=8
MOVL C00271 V=800.0 PL=8
MOVL C00272 V=800.0 PL=8
MOVL C00273 V=800.0 PL=8
MOVL C00274 V=800.0 PL=8
MOVL C00275 V=800.0 PL=8
MOVL C00276 V=800.0 PL=8
MOVL C00277 V=800.0 PL=8
MOVL C00278 V=800.0 PL=8
MOVL C00279 V=800.0 PL=8
MOVL C00280 V=800.0 PL=8
MOVL C00281 V=800.0 PL=0
SPYOF
MOVJ C00282 VJ=25.00 PL=0
SPYON
MOVL C00283 V=800.0 PL=8
MOVL C00284 V=800.0 PL=8
MOVL C00285 V=800.0 PL=8
MOVL C00286 V=800.0 PL=8
MOVL C00287 V=800.0 PL=8
MOVL C00288 V=800.0 PL=8
MOVL C00289 V=800.0 PL=8
MOVL C00290 V=800.0 PL=8
MOVL C00291 V=800.0 PL=8
MOVL C00292 V=800.0 PL=8
MOVL C00293 V=800.0 PL=8
MOVL C00294 V=800.0 PL=8
MOVL C00295 V=800.0 PL=8
MOVL C00296 V=800.0 PL=8
MOVL C00297 V=800.0 PL=8
MOVL C00298 V=800.0 PL=8
MOVL C00299 V=800.0 PL=8
MOVL C00300 V=800.0 PL=8
MOVL C00301 V=800.0 PL=8
MOVL C00302 V=800.0 PL=8
MOVL C00303 V=800.0 PL=8
MOVL C00304 V=800.0 PL=8
MOVL C00305 V=800.0 PL=8
MOVL C00306 V=800.0 PL=8
MOVL C00307 V=800.0 PL=8
MOVL C00308 V=800.0 PL=8
MOVL C00309 V=800.0 PL=8
MOVL C00310 V=800.0 PL=8
MOVL C00311 V=800.0 PL=0
SPYOF
MOVJ C00312 VJ=25.00 PL=0
SPYON
MOVL C00313 V=800.0 PL=8
MOVL C00314 V=800.0 PL=8
MOVL C00315 V=800.0 PL=8
MOVL C00316 V=800.0 PL=8
MOVL C00317 V=800.0 PL=8
MOVL C00318 V=800.0 PL=8
MOVL C00319 V=800.0 PL=8
MOVL C00320 V=800.0 PL=8
MOVL C00321 V=800.0 PL=8
MOVL C00322 V=800.0 PL=8
MOVL C00323 V=800.0 PL=8
MOVL C00324 V=800.0 PL=8
MOVL C00325 V=800.0 PL=8
MOVL C00326 V=800.0 PL=8
MOVL C00327 V=800.0 PL=8
MOVL C00328 V=800.0 PL=8
MOVL C00329 V=800.0 PL=8
MOVL C00330 V=800.0 PL=8
MOVL C00331 V=800.0 PL=8
MOVL C00332 V=800.0 PL=8
MOVL C00333 V=800.0 PL=8
MOVL C00334 V=800.0 PL=8
MOVL C00335 V=800.0 PL=8
MOVL C00336 V=800.0 PL=8
MOVL C00337 V=800.0 PL=8
MOVL C00338 V=800.0 PL=8
MOVL C00339 V=800.0 PL=8
MOVL C00340 V=800.0 PL=8
MOVL C00341 V=800.0 PL=8
MOVL C00342 V=800.0 PL=0
SPYOF
MOVJ C00343 VJ=25.00 PL=0
SPYON
MOVL C00344 V=800.0 PL=8
MOVL C00345 V=800.0 PL=8
MOVL C00346 V=800.0 PL=8
MOVL C00347 V=800.0 PL=8
MOVL C00348 V=800.0 PL=8
MOVL C00349 V=800.0 PL=8
MOVL C00350 V=800.0 PL=8
MOVL C00351 V=800.0 PL=8
MOVL C00352 V=800.0 PL=8
MOVL C00353 V=800.0 PL=8
MOVL C00354 V=800.0 PL=8
MOVL C00355 V=800.0 PL=8
MOVL C00356 V=800.0 PL=8
MOVL C00357 V=800.0 PL=8
MOVL C00358 V=800.0 PL=8
MOVL C00359 V=800.0 PL=8
MOVL C00360 V=800.0 PL=8
MOVL C00361 V=800.0 PL=8
MOVL C00362 V=800.0 PL=8
MOVL C00363 V=800.0 PL=8
MOVL C00364 V=800.0 PL=8
MOVL C00365 V=800.0 PL=8
MOVL C00366 V=800.0 PL=8
MOVL C00367 V=800.0 PL=8
MOVL C00368 V=800.0 PL=8
MOVL C00369 V=800.0 PL=8
MOVL C00370 V=800.0 PL=8
MOVL C00371 V=800.0 PL=8
MOVL C00372 V=800.0 PL=8
MOVL C00373 V=800.0 PL=8
MOVL C00374 V=800.0 PL=0
SPYOF
MOVJ C00375 VJ=25.00 PL=0
SPYON
MOVL C00376 V=800.0 PL=8
MOVL C00377 V=800.0 PL=8
MOVL C00378 V=800.0 PL=8
MOVL C00379 V=800.0 PL=8
MOVL C00380 V=800.0 PL=8
MOVL C00381 V=800.0 PL=8
MOVL C00382 V=800.0 PL=8
MOVL C00383 V=800.0 PL=8
MOVL C00384 V=800.0 PL=8
MOVL C00385 V=800.0 PL=8
MOVL C00386 V=800.0 PL=8
MOVL C00387 V=800.0 PL=8
MOVL C00388 V=800.0 PL=8
MOVL C00389 V=800.0 PL=8
MOVL C00390 V=800.0 PL=8
MOVL C00391 V=800.0 PL=8
MOVL C00392 V=800.0 PL=8
MOVL C00393 V=800.0 PL=8
MOVL C00394 V=800.0 PL=8
MOVL C00395 V=800.0 PL=8
MOVL C00396 V=800.0 PL=8
MOVL C00397 V=800.0 PL=8
MOVL C00398 V=800.0 PL=0
SPYOF
MOVJ C00399 VJ=25.00 PL=0
SPYON
MOVL C00400 V=800.0 PL=8
MOVL C00401 V=800.0 PL=8
MOVL C00402 V=800.0 PL=8
MOVL C00403 V=800.0 PL=8
MOVL C00404 V=800.0 PL=8
MOVL C00405 V=800.0 PL=8
MOVL C00406 V=800.0 PL=8
MOVL C00407 V=800.0 PL=8
MOVL C00408 V=800.0 PL=8
MOVL C00409 V=800.0 PL=8
MOVL C00410 V=800.0 PL=0
SPYOF
MOVJ C00411 VJ=25.00 PL=0
SPYON
MOVL C00412 V=800.0 PL=8
MOVL C00413 V=800.0 PL=8
MOVL C00414 V=800.0 PL=8
MOVL C00415 V=800.0 PL=8
MOVL C00416 V=800.0 PL=8
MOVL C00417 V=800.0 PL=8
MOVL C00418 V=800.0 PL=8
MOVL C00419 V=800.0 PL=8
MOVL C00420 V=800.0 PL=8
MOVL C00421 V=800.0 PL=8
MOVL C00422 V=800.0 PL=0
SPYOF
MOVJ C00423 VJ=25.00 PL=0
'Path End
MOVJ C00424 VJ=25.00 PL=0
END
